{attribute 'linkalways'} 
{attribute 'no_explicit_call' := 'This FB is a CLASS and must be accessed using methods or properties'}
{attribute 'enable_dynamic_creation'}
FUNCTION_BLOCK Node_F_VN_AppendToContainer_TcVnVector3_UINT EXTENDS VisionNode
VAR
    aElement : _TcVnVector3_UINT;
    ipContainer : _ITcVnContainer;
    hrPrev : _HRESULT(S_OK);
	hresult : _HRESULT(S_OK);
END_VAR

METHOD PUBLIC  Clone : I_Node
VAR
	pNode : POINTER TO Node_F_VN_AppendToContainer_TcVnVector3_UINT;
END_VAR
pNode := __NEW(Node_F_VN_AppendToContainer_TcVnVector3_UINT);
Clone := pNode^;
END_METHOD

METHOD FB_init : BOOL
VAR_INPUT
	bInitRetains : BOOL; // if TRUE, the retain variables are initialized (warm start / cold start)
	bInCopyCode : BOOL;  // if TRUE, the instance afterwards gets moved into the copy code (online change)
END_VAR
AddInput('aElement', aElement);
AddInput('ipContainer', ipContainer);
AddInput('hrPrev', hrPrev);
AddOutput('ipContainer', ipContainer);
AddOutput('hresult',hresult);
END_METHOD

METHOD PROTECTED OnExecute : HRESULT
hresult.Value := F_VN_AppendToContainer_TcVnVector3_UINT(
    aElement := aElement.Value,
	ipContainer := ipContainer.Value,
	hrPrev:= hrPrev.Value);
END_METHOD

METHOD PUBLIC PreExecutionCheck
VAR_INPUT
	Check : I_PreExecutionChecks;
END_VAR
Check.IsTrue(ipContainer.IsValid, 'ipContainer must be a valid container');
END_METHOD

END_FUNCTION_BLOCK

(* stored: Version 1.1.0.1, ProductVersion 3.1.4024.13
   POU Node_F_VN_AppendToContainer_TcVnVector3_UINT: Id {325aca21-015c-4ad7-9b9b-91439f54fe83}, SpecialFunc None
   Folder Constructor: Id {be8c8d1a-9c3a-4559-b35e-dc4823765653}
   Method Clone: Id {cf64125b-839c-4c56-b687-f392b018e786}
   Method FB_init: Id {8ef9292a-3926-4569-a586-dc7c44599974}
   Method OnExecute: Id {56215e73-8aa8-43cf-b880-23f8db27f276}
   Method PreExecutionCheck: Id {8f3ec1a0-f7f1-4b0f-9f76-05eb2ee84976} *)
